{attribute 'linkalways'} 
{attribute 'no_explicit_call' := 'This FB is a CLASS and must be accessed using methods or properties'}
{attribute 'enable_dynamic_creation'}
FUNCTION_BLOCK _Array0to3OfLREAL EXTENDS ArrayDatatypeBase
VAR CONSTANT
	lBound : DINT := 0;
	uBound : DINT := 3;
END_VAR
VAR
	localData : ARRAY [lBound..uBound] OF LREAL;
	activeData : REFERENCE TO ARRAY [lBound..uBound] OF LREAL REF= localData;
	elements : ARRAY [lBound..uBound] OF _LREAL(0.0);
	baseType : _LREAL(0.0);
END_VAR

PROPERTY PUBLIC Address : PVOID
GET
Address := ADR(activeData);
END_GET
END_PROPERTY

PROPERTY PUBLIC BaseDatatype : I_Datatype
GET
BaseDatatype := baseType;
END_GET
END_PROPERTY

METHOD PUBLIC ClearReference
VAR_INPUT
END_VAR
activeData REF= localData;
SetElementReference();
END_METHOD

METHOD PUBLIC Clone : I_Datatype
VAR
    pClone : POINTER TO _Array0to3OfLREAL;
END_VAR
pClone := __NEW(_Array0to3OfLREAL());
pClone^.Value := Value;
Clone := pClone^;
END_METHOD

METHOD FB_init : BOOL
VAR_INPUT
	bInitRetains : BOOL; // if TRUE, the retain variables are initialized (warm start / cold start)
	bInCopyCode : BOOL;  // if TRUE, the instance afterwards gets moved into the copy code (online change)
END_VAR
SetElementReference();
END_METHOD

METHOD PUBLIC GetElementAsDatatypeByIndex : I_Datatype
VAR_INPUT
	Index : DINT;
END_VAR
GetElementAsDatatypeByIndex := elements[Index];
END_METHOD

METHOD PUBLIC GetElementByIndex : REFERENCE TO _LREAL;
VAR_INPUT
	Index : DINT;
END_VAR
GetElementByIndex REF= elements[Index];
END_METHOD

PROPERTY PUBLIC LowerBound : DINT
GET
LowerBound := lBound;
END_GET
END_PROPERTY

METHOD PUBLIC MakeReferenceTo
VAR_INPUT
	ReferenceTarget : REFERENCE TO ARRAY [lBound..uBound] OF LREAL;
END_VAR
activeData REF= ReferenceTarget;
SetElementReference();
END_METHOD

METHOD PROTECTED OnSerializeArrayValues
VAR_INPUT
	Serializer : I_Serializer;
END_VAR
VAR
	i : DINT;
END_VAR
FOR i := lBound TO uBound DO
	elements[i].SerializeWith(Serializer);
END_FOR
END_METHOD

METHOD PROTECTED SetElementReference
VAR_INPUT
END_VAR
VAR
	i : DINT;
END_VAR
FOR i := lBound TO uBound DO
	elements[i].MakeReferenceTo(activeData[i]);
END_FOR
END_METHOD

PROPERTY PUBLIC Size : UDINT
GET
Size := SIZEOF(activeData);
END_GET
END_PROPERTY

METHOD PROTECTED TryDeserializeArrayValues : BOOL
VAR_INPUT
	Deserializer : I_Deserializer;
	Feedback : I_DeserializerFeedback;
END_VAR
VAR
	enumerator : I_DeserializerArrayForwardEnumerator;
	i : DINT;
END_VAR
enumerator := Deserializer.GetArrayEnumerator();
i := lBound;

WHILE enumerator.MoveNext() AND i <= uBound DO
	
	IF NOT elements[i].TryDeserializeFrom(enumerator.Current, Feedback) THEN
		EXIT;
	END_IF
	i := i + 1;

END_WHILE
enumerator.Dispose();
END_METHOD

METHOD TryMakeReferenceTo : BOOL
VAR_INPUT
	Target : I_Datatype;
END_VAR
VAR
	targetAsArray : I_ArrayDatatype;
	pTargetData : POINTER TO ARRAY [lBound..uBound] OF LREAL;
END_VAR
IF NOT Target.TryResolveAsArrayDatatype(targetAsArray) THEN
	RETURN;
END_IF

IF NOT (targetAsArray.Identifier = Identifier) THEN
	RETURN;
END_IF

pTargetData := Target.Address;
activeData REF= pTargetData^;
SetElementReference();
TryMakeReferenceTo := TRUE;
END_METHOD

PROPERTY PUBLIC UpperBound : DINT
GET
UpperBound := ubound;
END_GET
END_PROPERTY

PROPERTY PUBLIC Value : REFERENCE TO ARRAY [lBound..uBound] OF LREAL;
GET
Value ref= activeData;
END_GET
END_PROPERTY

END_FUNCTION_BLOCK

(* stored: Version 1.1.0.1, ProductVersion 3.1.4024.13
   POU _Array0to3OfLREAL: Id {88ad166a-5397-07f4-22ee-a9d032ff2e42}, SpecialFunc None
   Folder Core: Id {c14478c1-e2d0-0d41-24c4-c830c47b44de}
   Folder Constructor: Id {33774c7b-4121-053f-37ba-bd0d99ee8d32}
   Folder Protected: Id {8e31f85b-8fb2-0d56-39c8-9ed62de3b7f0}
   Folder Customize: Id {ee87abc0-c851-0395-2add-d49f3e4b5077}
   Property Address: Id {01f05dd5-01be-0e35-0db6-9185c1ea1a31}
   Get Get: Id {b946089f-327a-0a2c-14d8-63ec39fafc77}
   Property BaseDatatype: Id {b0136d28-1ba2-0e3e-3699-3bb3cbfc9437}
   Get Get: Id {d172eb44-c0f8-0c76-0d31-1c1b692bfccb}
   Method ClearReference: Id {7927049b-6aa2-011b-194c-4a208e398203}
   Method Clone: Id {079c774f-aaac-0fb4-32fe-d081d068b2e5}
   Method FB_init: Id {1e37f82a-34fc-0ffa-2b43-167e42156956}
   Method GetElementAsDatatypeByIndex: Id {ee79bb66-39e8-0032-18f7-835240fc1532}
   Method GetElementByIndex: Id {e7dcf353-d686-08a7-1f84-29529cb0934c}
   Property LowerBound: Id {57df1dc7-457c-0672-1c9e-5323c3b95b40}
   Get Get: Id {b90c51d8-8241-0e02-3985-ee1b40f08357}
   Method MakeReferenceTo: Id {b2246a5e-2e90-037f-0e0e-171a759910d8}
   Method OnSerializeArrayValues: Id {94f2c2c4-8723-04e6-3293-ce67d5069e97}
   Method SetElementReference: Id {81665e1e-5b4e-0164-3d8e-7a8d5d049301}
   Property Size: Id {845f6342-0a17-0348-1830-4c94b6a85b39}
   Get Get: Id {0dae24ca-b30d-05b4-1406-8a5929740ab7}
   Method TryDeserializeArrayValues: Id {d9e218bb-62e3-0566-225e-a19430eaa386}
   Method TryMakeReferenceTo: Id {e8809a01-c70d-03fa-13d2-d2b40ef633b7}
   Property UpperBound: Id {f857e726-9d64-07c0-0019-43f2986fd483}
   Get Get: Id {0131df47-9b38-0d36-1665-b90769689be8}
   Property Value: Id {048d3ffa-fe89-077a-2778-756342378518}
   Get Get: Id {14d5e013-452e-0432-12fe-9f722e04cb9d} *)
